SUBAPPLICATION Uebung_077_AUI (* RHS Position/Force/Draft auf UT ausgeben mit AR_Timeout_Zero (Adapter Version) *)
  (* Standard: 61499-2; Description: Copyright (c) 2026 Meisterschulen am Ostbahnhof This program and the accompanying materials are made available under the terms of the Eclipse Public License 2.0 which is available at https://www.eclipse.org/legal/epl-2.0/ SPDX-License-Identifier: EPL-2.0 *)
  (* Version 1.0, 2026-09-17, Franz Höpfinger, Meisterschulen am Ostbahnhof, ISOBUS TECU Rear Hitch Status (RHS): Position/Force/Draft mit AR_Timeout_Zero Fendt-Schaltung auf UT ausgeben (Adapter Version, analog Krauternter TECU_RHS.SUB) *)
  PACKAGE Uebungen;
  IMPORT Uebungen::const::UT::TECU::DefaultPool_TECU_Numeric::NumberVariable_TECU_RHS_Position_N;
  IMPORT Uebungen::const::UT::TECU::DefaultPool_TECU_Numeric::NumberVariable_TECU_RHS_Force_N;
  IMPORT Uebungen::const::UT::TECU::DefaultPool_TECU_Numeric::NumberVariable_TECU_RHS_Draft_N;
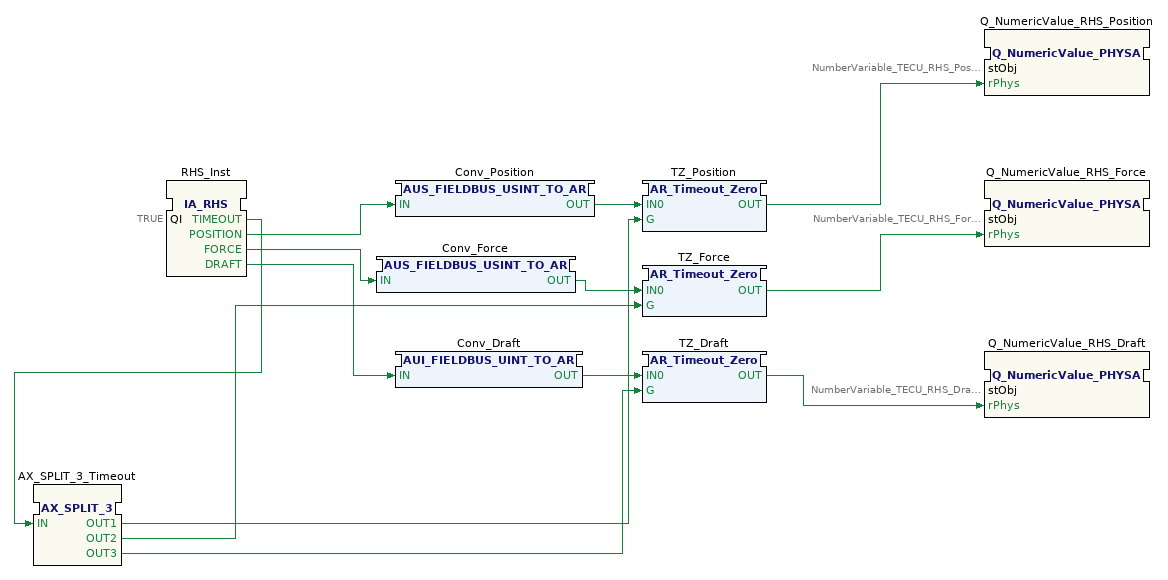
  FBS
    RHS_Inst : isobus::tecu::IA_RHS(QI := TRUE);
    Q_NumericValue_RHS_Position : isobus::UT::Q::Q_NumericValue_PHYSA(stObj := NumberVariable_TECU_RHS_Position_N);
    Q_NumericValue_RHS_Force : isobus::UT::Q::Q_NumericValue_PHYSA(stObj := NumberVariable_TECU_RHS_Force_N);
    Q_NumericValue_RHS_Draft : isobus::UT::Q::Q_NumericValue_PHYSA(stObj := NumberVariable_TECU_RHS_Draft_N);
    AX_SPLIT_3_Timeout : adapter::events::unidirectional::AX_SPLIT_3;
  END_FBS
  SUBAPPS
    Conv_Position : MyLib::sys::AUS_FIELDBUS_USINT_TO_AR;
    TZ_Position : MyLib::sys::AR_Timeout_Zero;
    Conv_Force : MyLib::sys::AUS_FIELDBUS_USINT_TO_AR;
    TZ_Force : MyLib::sys::AR_Timeout_Zero;
    Conv_Draft : MyLib::sys::AUI_FIELDBUS_UINT_TO_AR;
    TZ_Draft : MyLib::sys::AR_Timeout_Zero;
  END_SUBAPPS
  ADAPTER_CONNECTIONS
    RHS_Inst.TIMEOUT TO AX_SPLIT_3_Timeout.IN;
    RHS_Inst.POSITION TO Conv_Position.IN;
    Conv_Position.OUT TO TZ_Position.IN0;
    AX_SPLIT_3_Timeout.OUT1 TO TZ_Position.G;
    TZ_Position.OUT TO Q_NumericValue_RHS_Position.rPhys;
    RHS_Inst.FORCE TO Conv_Force.IN;
    Conv_Force.OUT TO TZ_Force.IN0;
    AX_SPLIT_3_Timeout.OUT2 TO TZ_Force.G;
    TZ_Force.OUT TO Q_NumericValue_RHS_Force.rPhys;
    RHS_Inst.DRAFT TO Conv_Draft.IN;
    Conv_Draft.OUT TO TZ_Draft.IN0;
    AX_SPLIT_3_Timeout.OUT3 TO TZ_Draft.G;
    TZ_Draft.OUT TO Q_NumericValue_RHS_Draft.rPhys;
  END_CONNECTIONS
END_SUBAPPLICATION
